FUNCTION_BLOCK FB_CheckWeigher EXTENDS FB_Station
VAR_INPUT
END_VAR
VAR_OUTPUT
END_VAR
VAR
	bTriggerRead			AT %Q* : BOOL;
	sBarcodeRead			AT %I* : STRING(255);
	iWorkState				: DINT;
	iRetries				: DINT;
	tmrRetry				: TON;
END_VAR
VAR CONSTANT
	NO_READ					: STRING(255) := 'NO_READ';
	READ_RETRY_COUNT		: DINT := 3;
END_VAR

METHOD PROTECTED  DoWork : BOOL
VAR_INPUT
END_VAR
CASE iWorkState OF
	0:
		iRetries := 0;
		sBarcodeRead := '';
		iWorkState := 10;
		bTriggerRead := TRUE;
		
	10:
		IF sBarcodeRead <> '' THEN
			bTriggerRead := FALSE;
			iWorkState := 20;
		END_IF
		
	11:
		tmrRetry(IN:=TRUE, PT:=T#500MS);
		IF tmrRetry.Q THEN
			tmrRetry(IN:=FALSE);
			bTriggerRead := TRUE;
			iWorkState := 20;
		END_IF
		
	20:
		IF sBarcodeRead = NO_READ THEN
			IF iRetries < READ_RETRY_COUNT THEN
				iRetries := iRetries + 1;
				iWorkState := 11;
			ELSE
				pPartStatus^.bBarcodeStatus := FALSE;
				pPartStatus^.sBarcode := NO_READ;
				iWorkState := 30;
			END_IF
		ELSE
			pPartStatus^.bBarcodeStatus := TRUE;
			pPartStatus^.sBarcode := sBarcodeRead;
			iWorkState := 30;
		END_IF
		
	30:
		iWorkState := 0;
		DoWork := TRUE;
	
END_CASE
END_METHOD

METHOD PROTECTED  FaultHandler : E_StationState
VAR_INPUT
END_VAR
END_METHOD

END_FUNCTION_BLOCK

(* stored: Version 1.1.0.1, ProductVersion 3.1.4024.12
   POU FB_CheckWeigher: Id {f2b6ec40-0a7e-498d-ad24-1bc64cb8a48b}, SpecialFunc None
   Method DoWork: Id {06478269-7e8f-4cf3-8ab9-628ebb68d97b}
   Method FaultHandler: Id {f883c496-e31b-4a3f-bc0d-333d136fe914} *)
